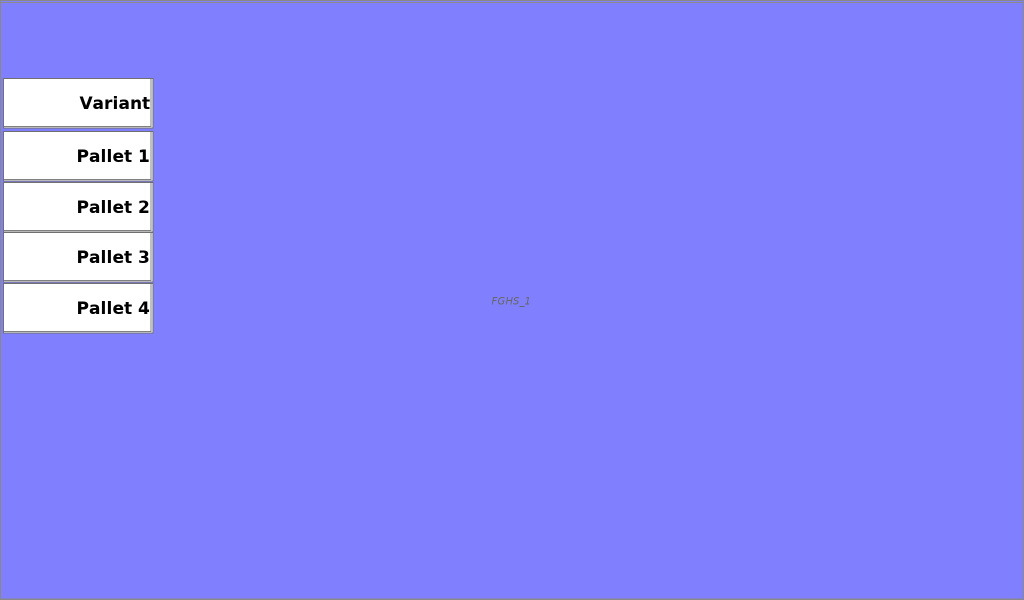
VISUALIZATION FGHS  // 1024x600
    Frame (0,2 1023x598)
        shows FGHS_1()
        shows DataPallet1()
        shows DataPallet2()
        shows DataPallet3()
        shows DataPallet4()
    Button (3,78 150x50), "Variant", image: VisuSymbols.Symbols.Database2
        OnMouseDown: FrameSelectionChange Selection=SelectedFrame=146e207b-fd78-4676-ba16-384fa245d7d2, GlobSel=AssignDir=MainPage.GenElemInst_1003, AssignType=Directly, SelType=Locally
    Button (3,131 150x50), "Pallet 1", image: VisuSymbols.Symbols.Database2
        OnMouseDown: FrameSelectionChange Selection=SelectedFrame=146e207b-fd78-4676-ba16-384fa245d7d2, Selection=1, GlobSel=AssignDir=MainPage.GenElemInst_1003, AssignType=Directly, SelType=Locally
    Button (3,182 150x50), "Pallet 2", image: VisuSymbols.Symbols.Database2
        OnMouseDown: FrameSelectionChange Selection=SelectedFrame=146e207b-fd78-4676-ba16-384fa245d7d2, Selection=2, GlobSel=AssignDir=MainPage.GenElemInst_1003, AssignType=Directly, SelType=Locally
    Button (3,232 150x50), "Pallet 3", image: VisuSymbols.Symbols.Database2
        OnMouseDown: FrameSelectionChange Selection=SelectedFrame=146e207b-fd78-4676-ba16-384fa245d7d2, Selection=3, GlobSel=AssignDir=MainPage.GenElemInst_1003, AssignType=Directly, SelType=Locally
    Button (3,283 150x50), "Pallet 4", image: VisuSymbols.Symbols.Database2
        OnMouseDown: FrameSelectionChange Selection=SelectedFrame=146e207b-fd78-4676-ba16-384fa245d7d2, Selection=4, GlobSel=AssignDir=MainPage.GenElemInst_1003, AssignType=Directly, SelType=Locally
END_VISUALIZATION

(* stored: Version 1.1.0.1, ProductVersion 3.1.4024.12
   Visu FGHS: Id {ce414ec2-39b0-480f-81ae-b8e8993e9803} *)
